// TIA Portal V16 export
// export: Created 2022-04-14T22:41:07.0074403Z, ExportSetting WithDefaults, DisplayName Totally Integrated Automation Portal, DisplayVersion V16, DisplayName TIA Portal Version Control Interface, DisplayVersion V16, DisplayName TIA Portal Openness, DisplayVersion V16, DisplayName STEP 7 Professional, DisplayVersion V16, DisplayName STEP 7 Safety, DisplayVersion V16, DisplayName WinCC Professional, DisplayVersion V16
VAR_GLOBAL   // PLC tag table "Standard-Variablentabelle"
   "Auto/Manual" AT %I0.0 : Bool;
   Start AT %I0.1 : Bool;
   Reset AT %I0.2 : Bool;
   Stop AT %I0.3 : Bool;
   Estop AT %I0.4 : Bool;
   "Conveyor Sensor 1" AT %I0.5 : Bool;
   "Conveyor Sensor 2" AT %I0.6 : Bool;
   "Conveyor Sensor 3" AT %I0.7 : Bool;
   "Alarm Siren" AT %Q0.0 : Bool;
   "Start Light" AT %Q0.1 : Bool;
   "Reset Light" AT %Q0.2 : Bool;
   "Stop Light" AT %Q0.3 : Bool;
   "Pusher 2" AT %Q0.5 : Bool;
   "Stack Light Green" AT %Q0.6 : Bool;
   "Stack Light Yellow" AT %Q0.7 : Bool;
   "Ready to Run" AT %M0.0 : Bool;
   "Reset Memory" AT %M0.5 : Bool;
   "Pusher Sensor 1 Mem" AT %M0.6 : Bool;
   "Pusher 1 FW Mem" AT %M0.7 : Bool;
   "Pusher Sensor 2 Mem" AT %M1.0 : Bool;
   "Pusher 2 FW Mem" AT %M1.1 : Bool;
   "Conveyor Sensor 4" AT %I1.0 : Bool;
   "Pusher Sensor 1" AT %I1.1 : Bool;
   "Pusher Sensor 2" AT %I1.2 : Bool;
   "Pusher 1 FW" AT %I1.3 : Bool;
   "Pusher 2 FW" AT %I1.4 : Bool;
   "Pusher 1" AT %Q0.4 : Bool;
   "Stack Light Red" AT %Q1.0 : Bool;
   "Drain 1" AT %Q1.1 : Bool;
   "Drain 2" AT %Q1.2 : Bool;
   "Drain 3" AT %Q1.3 : Bool;
   "Conveyor 1" AT %QW36 : Int;
   "Conveyor 2" AT %Q1.5 : Bool;
   "Conveyor 3" AT %Q1.6 : Bool;
   "Conveyor 4" AT %Q1.7 : Bool;
   "Conveyor Sensor 1 Mem" AT %M1.2 : Bool;
   "Conveyor Sensor 2 Mem" AT %M1.3 : Bool;
   "Conveyor Sensor 3 Mem" AT %M1.4 : Bool;
   "Conveyor Sensor 4 Mem" AT %M1.5 : Bool;
   "Conveyor Sensor 5 Mem" AT %M1.6 : Bool;
   "Advanced Feeder" AT %Q2.1 : Bool;
   "Conveyor Sensor 5" AT %I1.5 : Bool;
   "Running Torque" AT %IW30 : Int;
   "Running Temperature" AT %IW32 : Int;
   "Error Message" AT %Q2.2 : Bool;
   "1.5 KG" AT %QW30 : Int;
   "5.0 KG" AT %QW32 : Int;
   "7.5" AT %QW34 : Int;
   "Estop Memory" AT %M0.1 : Bool;
END_VAR
